PROGRAM MAIN
VAR
	nState: INT;
	bButton	:	BOOL;
	fbMotion	:	FB_Motion;
	T1: TON;
END_VAR



stAxis1.IN.bPower	:=	TRUE;
stAxis1.IN.fOverride	:=	100;

fbMotion(Axis:=Axis1 , staxisinterface:=stAxis1 );
ACT_Motion();

ACTION ACT_Motion:
CASE nState OF 
	

	0:
	
		IF bButton AND NOT stAxis1.OUT.bPowerErr
		AND stAxis1.OUT.bPowerEnabled
		AND NOT stAxis1.OUT.bPowerErr 
		AND	NOT stAxis1.OUT.bStopActive THEN
		
			nState := 10;
		
		END_IF
		
		
	10:
	
	stAxis1.IN.bMoveAbs	:=	TRUE;
	stAxis1.IN.bStop	:=	FALSE;	
	
	stAxis1.IN.fPosition	:=	1000;
	stAxis1.IN.fVelocity	:=	500;
	
	IF stAxis1.OUT.bMoveAbsBusy 
	AND NOT stAxis1.OUT.bMoveAbsErr
	AND NOT	stAxis1.OUT.bMoveAbsErr	THEN	
	
		nState := 20;	
	
	ELSIF stAxis1.OUT.bMoveAbsErr THEN
		
		nState:=999;
		
	END_IF
	
	
	20:
	
	IF  stAxis1.OUT.bMoveAbsDone 
	AND NOT stAxis1.OUT.bMoveAbsErr THEN

		stAxis1.IN.bMoveAbs:=FALSE;
		nState:=25;	
		
		
	ELSIF stAxis1.OUT.bMoveAbsErr THEN
		
		nState := 999;
	
	END_IF
	
	
	25:
	
	T1(IN:=TRUE , PT:=T#5S, Q=> , ET=> );
	
	IF T1.Q THEN
		nState := 30;
	T1(IN:=TRUE);
	END_IF

	30:
	
	stAxis1.IN.bMoveAbs	:=	TRUE;
	stAxis1.IN.bStop	:=	FALSE;	
	
	stAxis1.IN.fPosition	:=	5000;
	stAxis1.IN.fVelocity	:=	750;
	
	IF stAxis1.OUT.bMoveAbsBusy 
	AND NOT stAxis1.OUT.bMoveAbsErr
	AND NOT	stAxis1.OUT.bMoveAbsErr	THEN	
	
		nState := 40;	
	
	ELSIF stAxis1.OUT.bMoveAbsErr THEN
		
		nState:=999;
		
	END_IF
	
	
	40:
	
	IF  stAxis1.OUT.bMoveAbsDone 
	AND NOT stAxis1.OUT.bMoveAbsErr THEN

		stAxis1.IN.bMoveAbs:=FALSE;
		nState	:=	50;	
		
		
	ELSIF stAxis1.OUT.bMoveAbsErr THEN
		
		nState := 999;
	
	END_IF
	
	
	50:
	
	stAxis1.IN.bMoveAbs	:=	TRUE;
	stAxis1.IN.bStop	:=	FALSE;	
	
	stAxis1.IN.fPosition	:=	0;
	stAxis1.IN.fVelocity	:=	1000;
	
	IF stAxis1.OUT.bMoveAbsBusy 
	AND NOT stAxis1.OUT.bMoveAbsErr
	AND NOT	stAxis1.OUT.bMoveAbsErr	THEN	
	
		nState := 60;	
	
	ELSIF stAxis1.OUT.bMoveAbsErr THEN
		
		nState:=999;
		
	END_IF
	
	
	60:
	
	IF  stAxis1.OUT.bMoveAbsDone 
	AND NOT stAxis1.OUT.bMoveAbsErr THEN

		stAxis1.IN.bMoveAbs:=FALSE;
		nState	:=	0;	
		
		
	ELSIF stAxis1.OUT.bMoveAbsErr THEN
		
		nState := 999;
	
	END_IF
	
	
	
	
END_CASE
END_ACTION

END_PROGRAM

(* stored: Version 1.1.0.1, ProductVersion 3.1.4024.4
   POU MAIN: Id {42c2396e-1ffd-4478-a301-53d386c26b32}, SpecialFunc None
   Action ACT_Motion: Id {538727a7-876b-4a14-b34e-503c6999e632} *)
